(* IEC 61131-3 sources: repolevel_ST_code_completion/dataset/project_code/SRCI-main/PRG, 3 files *)

(* ---- Example_ChangeSpeedOverride.st ---- *)
PROGRAM Example_ChangeSpeedOverride
VAR_INPUT
  /// Start command execution
  Execute : BOOL;
  /// Command parameter
  ParCmd  : ChangeSpeedOverrideParCmd;
END_VAR

VAR_OUTPUT
  /// Error ID
  ErrorID     : DINT;
  /// Error addition text
  ErrorAddTxt : STRING;
  /// Command outputs
  OutCmd      : ChangeSpeedOverrideOutCmd;
END_VAR

VAR
  /// internal step counter
 _stepCmd    : DINT;
  /// internal timer for command
 _timerCmd   : TON;
  /// internal timeout for command
 _timeoutCmd : TIME := T#5S;
END_VAR

// forwarding command parameter(s)
ChangeSpeedOverride.ParCmd := ParCmd;
// forwarding command output(s)
OutCmd := ChangeSpeedOverride.OutCmd;

CASE _stepCmd OF

  0: // start execution ?
     IF ( Execute )
     THEN
       // Reset request
       Execute := FALSE;
       // set timeout
       SetTimeout(PT := _timeoutCmd, rTimer := _timerCmd);
       // inc step counter
      _stepCmd := _stepCmd + 1;
     END_IF

  1: // Start Execution
     IF (( NOT ChangeSpeedOverride.Error  ) AND
         ( NOT ChangeSpeedOverride.Error  ))
     THEN
       // start execution
       SetSequence.Execute := TRUE;
       // set timeout
       SetTimeout(PT := _timeoutCmd, rTimer := _timerCmd);
       // inc step counter
      _stepCmd := _stepCmd + 1;
     ELSE
       // timeout exceeded ?
       IF (CheckTimeout(_timerCmd) = RobotLibraryConstants.OK)
       THEN
         ErrorID     := RobotLibraryErrorIdEnum.ERR_TIMEOUT_CMD;
         ErrorAddTxt := CONCAT('_stepCmd = ' , DINT_TO_STRING(_stepCmd));
       END_IF

       // Error occurred ?
       IF (ChangeSpeedOverride.Error)
       THEN
         ErrorID     := ChangeSpeedOverride.ErrorID;
         ErrorAddTxt := CONCAT('_stepCmd = ' , DINT_TO_STRING(_stepCmd));
       END_IF
     END_IF

  2: // Wait Execution done ?
     IF (( NOT ChangeSpeedOverride.Busy ) AND
         (     ChangeSpeedOverride.Done ))
     THEN
       // stop execution
       ChangeSpeedOverride.Execute := FALSE;
       // set timeout
       SetTimeout(PT := _timeoutCmd, rTimer := _timerCmd);
       // set step counter
      _stepCmd := 0;
     ELSE
       // timeout exceeded ?
       IF (CheckTimeout(_timerCmd) = RobotLibraryConstants.OK)
       THEN
         ErrorID     := RobotLibraryErrorIdEnum.ERR_TIMEOUT_CMD;
         ErrorAddTxt := CONCAT('_stepCmd = ' , DINT_TO_STRING(_stepCmd));
       END_IF

       // Error occurred ?
       IF (ChangeSpeedOverride.Error)
       THEN
         ErrorID     := ChangeSpeedOverride.ErrorID;
         ErrorAddTxt := CONCAT('_stepCmd = ' , DINT_TO_STRING(_stepCmd));
       END_IF
     END_IF

ELSE
  // invalid step
  ErrorID     := RobotLibraryErrorIdEnum.ERR_INVALID_STEP;
  ErrorAddTxt := CONCAT('_stepCmd = ' , DINT_TO_STRING(_stepCmd));
END_CASE

// Call functionblock
ChangeSpeedOverride
(
  Name         := 'ChangeSpeedOverride',
  ExecMode     := ExecutionMode.PARALLEL,
  Priority     := PriorityLevel.NORMAL,
  AxesGroup    := AxesGroup
);

(* ---- Example_EnableRobot.st ---- *)
PROGRAM Example_EnableRobot
VAR_INPUT
  /// Enable command
  Enable : BOOL;
  /// Command parameter
  ParCmd : EnableRobotParCmd;
END_VAR

VAR_OUTPUT
  /// Error ID
  ErrorID     : DINT;
  /// Error addition text
  ErrorAddTxt : STRING;
  /// Command outputs
  OutCmd      : EnableRobotOutCmd;
END_VAR

VAR
  /// internal step counter
 _stepCmd    : DINT;
  /// internal timer for command
 _timerCmd   : TON;
  /// internal timeout for command
 _timeoutCmd : TIME := T#5S;
END_VAR

// forwarding command parameter(s) / command outputs
EnableRobot.ParCmd := ParCmd;
// forwarding command output(s)
OutCmd := EnableRobot.OutCmd;

CASE _stepCmd OF

  0: // Enable or disable function ?
     IF (( Enable           ) XOR
         ( UserData.Enabled ))
     THEN
       // set timeout
       SetTimeout(PT := _timeoutCmd, rTimer := _timerCmd);
       // inc step counter
      _stepCmd := _stepCmd + 1;
     END_IF

  1: // Start Execution
     IF (( NOT EnableRobot.Busy  ) AND
         ( NOT EnableRobot.Error ))
     THEN
       // enable/disable robot
       EnableRobot.Enable := Enable;
       // set timeout
       SetTimeout(PT := _timeoutCmd, rTimer := _timerCmd);
       // inc step counter
      _stepCmd := _stepCmd + 1;
     ELSE
       // timeout exceeded ?
       IF (CheckTimeout(_timerCmd) = RobotLibraryConstants.OK)
       THEN
         ErrorID     := RobotLibraryErrorIdEnum.ERR_TIMEOUT_CMD;
         ErrorAddTxt := CONCAT('_stepCmd = ' , DINT_TO_STRING(_stepCmd));
       END_IF

       // Error occurred ?
       IF (EnableRobot.Error)
       THEN
         ErrorID     := EnableRobot.ErrorID;
         ErrorAddTxt := CONCAT('_stepCmd = ' , DINT_TO_STRING(_stepCmd));
       END_IF
     END_IF

  2: // Wait Execution done ?
     IF (( NOT EnableRobot.Error            ) AND
         (     EnableRobot.Enabled = Enable ))
     THEN
       // set timeout
       SetTimeout(PT := _timeoutCmd, rTimer := _timerCmd);
       // set step counter
      _stepCmd := 0;
     ELSE
       // timeout exceeded ?
       IF (CheckTimeout(_timerCmd) = RobotLibraryConstants.OK)
       THEN
         ErrorID     := RobotLibraryErrorIdEnum.ERR_TIMEOUT_CMD;
         ErrorAddTxt := CONCAT('_stepCmd = ' , DINT_TO_STRING(_stepCmd));
       END_IF

       // Error occurred ?
       IF (EnableRobot.Error)
       THEN
         ErrorID     := EnableRobot.ErrorID;
         ErrorAddTxt := CONCAT('_stepCmd = ' , DINT_TO_STRING(_stepCmd));
       END_IF
     END_IF

ELSE
  // invalid step
  ErrorID     := RobotLibraryErrorIdEnum.ERR_INVALID_STEP;
  ErrorAddTxt := CONCAT('_stepCmd = ' , DINT_TO_STRING(_stepCmd));
END_CASE

// call function block
EnableRobot
(
  Name      := 'EnableRobot',
  ExecMode  := ExecutionMode.PARALLEL,
  Priority  := PriorityLevel.NORMAL,
  AxesGroup := AxesGroup,
);

(* ---- Example_GroupContinue.st ---- *)
PROGRAM Example_GroupContinue
VAR_INPUT
  /// Start command execution
  Execute : BOOL;
END_VAR

VAR_OUTPUT
  /// Error ID
  ErrorID     : DINT;
  /// Error addition text
  ErrorAddTxt : STRING;
END_VAR

VAR
  /// internal step counter
 _stepCmd    : DINT;
  /// internal timer for command
 _timerCmd   : TON;
  /// internal timeout for command
 _timeoutCmd : TIME := T#5S;
END_VAR

CASE _stepCmd OF

  0: // start execution ?
     IF ( Execute )
     THEN
       // reset request
       Execute := FALSE;
       // set timeout
       SetTimeout(PT := _timeoutCmd, rTimer := _timerCmd);
       // inc step counter
      _stepCmd := _stepCmd + 1;
     END_IF

  1: // Start Execution
     IF (( NOT GroupContinue.Busy  ) AND
         ( NOT GroupContinue.Error ))
     THEN
       // start execution
       GroupContinue.Execute := TRUE;
       // set timeout
       SetTimeout(PT := _timeoutCmd, rTimer := _timerCmd);
       // inc step counter
      _stepCmd := _stepCmd + 1;
     ELSE
       // timeout exceeded ?
       IF (CheckTimeout(_timerCmd) = RobotLibraryConstants.OK)
       THEN
         ErrorID     := RobotLibraryErrorIdEnum.ERR_TIMEOUT_CMD;
         ErrorAddTxt := CONCAT('_stepCmd = ' , DINT_TO_STRING(_stepCmd));
       END_IF

       // Error occurred ?
       IF (GroupContinue.Error)
       THEN
         ErrorID     := GroupContinue.ErrorID;
         ErrorAddTxt := CONCAT('_stepCmd = ' , DINT_TO_STRING(_stepCmd));
       END_IF
     END_IF

  2: // Wait Execution done ?
     IF (( NOT GroupContinue.Error ) AND
         (     GroupContinue.Done  ))
     THEN
       // stop execution
       GroupContinue.Execute := FALSE;
       // set timeout
       SetTimeout(PT := _timeoutCmd, rTimer := _timerCmd);
       // set step counter
      _stepCmd := 0;
     ELSE
       // timeout exceeded ?
       IF (CheckTimeout(_timerCmd) = RobotLibraryConstants.OK)
       THEN
         ErrorID     := RobotLibraryErrorIdEnum.ERR_TIMEOUT_CMD;
         ErrorAddTxt := CONCAT('_stepCmd = ' , DINT_TO_STRING(_stepCmd));
       END_IF

       // Error occurred ?
       IF (GroupContinue.Error)
       THEN
         ErrorID     := GroupContinue.ErrorID;
         ErrorAddTxt := CONCAT('_stepCmd = ' , DINT_TO_STRING(_stepCmd));
       END_IF
     END_IF

ELSE
  // invalid step
  ErrorID     := RobotLibraryErrorIdEnum.ERR_INVALID_STEP;
  ErrorAddTxt := CONCAT('_stepCmd = ' , DINT_TO_STRING(_stepCmd));
END_CASE

// call function block
GroupContinue
(
  Name      := 'GroupContinue',
  ExecMode  := ExecutionMode.PARALLEL,
  Priority  := PriorityLevel.NORMAL,
  AxesGroup := AxesGroup
);
